TYPE TestStruct2 :
STRUCT
	bTest			: BOOL := TRUE;
	fTestLreal		: LREAL := 77.777;
	sTest			: T_MAXSTRING := 'This could be a really long string...';
	//aInt			: ARRAY[0..2] OF INT;
END_STRUCT
END_TYPE

(* stored: Version 1.1.0.1, ProductVersion 3.1.4024.6
   DUT TestStruct2: Id {4d41ed42-484f-4ec3-8dfc-b65924c5a5e7} *)
